PROGRAM MAIN
VAR
	SealedinCoil: FbSealedinCoil;
	xTrigger: BOOL;
	xSealedInCoil: BOOL;
	StateCoilFaultCoil: FbStateCoilFaultCoil;
	xBreakCondition: BOOL;
	xMemoryCoil: BOOL;
	StartStopCircuit: FbStartStopCircuit;
	xStart: BOOL;
	xStop: BOOL;
	/// use SR instead 
	SetReset: FbSetReset;
	xRun: BOOL;
	xSet: BOOL;
	/// use RS instead 
	ResetSet: FbResetSet;
	xReset: BOOL;
	xQs: BOOL;
	xQr: BOOL;
	/// use BLINK instead 
	Flasher: FbFlasher;
	xFlashingLight: BOOL;
	Debounce: FbDebounce;
	xInput: BOOL;
	xInputDebounced: BOOL;
	ExtendCylinder: fbStep;
	xExtendCylinderCmd: BOOL;
	TONExtendCylinderDone: TON;
	xExtendCylinderDone: BOOL;
	tETExtend: TIME;
	RetractCylinder: fbStep;
	xRetractCylinderCmd: BOOL;
	TONRetractCylinderDone: TON;
	tETRetract: TIME;
	Mission: FbMission;
	xMission1Start: BOOL;
	xMission2Start: BOOL;
	xMission1Done: BOOL;
	xMission2Done: BOOL;
	xNoMission: BOOL;
	xMission1Busy: BOOL;
	xMission2Busy: BOOL;
	FiveRung: fbFiveRung;
	xFromSeqLogic: BOOL;
	xEStopOK: BOOL;
	xAutoMode: BOOL;
	xManMode: BOOL;
	xPushButton: BOOL;
	xSensor: BOOL;
	xResetFault: BOOL;
	xTriggerf: BOOL;
	xSafe: BOOL;
	xCommand: BOOL;
	xInPosition: BOOL;
	xTimeoutFault: BOOL;
	Mode: FbMode;
	xAutoModePB: BOOL;
	xManModePB: BOOL;
	xAutoSelected: BOOL;
	xManualSelected: BOOL;
END_VAR

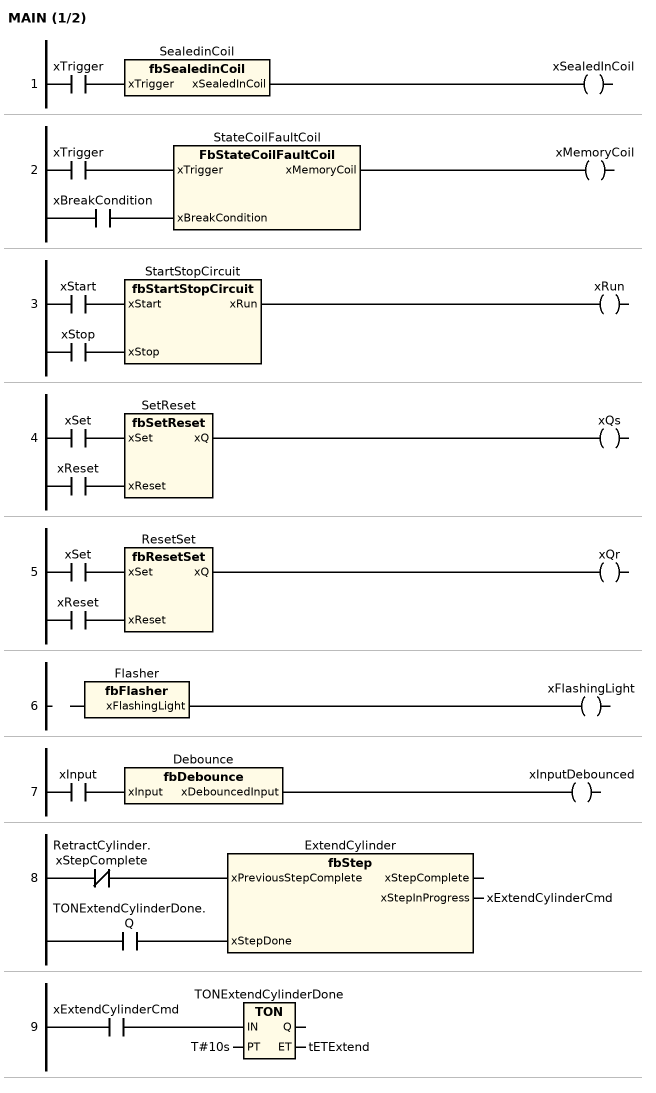
// NETWORK 1
SealedinCoil(xTrigger := xTrigger); // fbSealedinCoil
xSealedInCoil := SealedinCoil.xSealedInCoil;

// NETWORK 2
StateCoilFaultCoil(xTrigger := xTrigger, xBreakCondition := xBreakCondition); // FbStateCoilFaultCoil
xMemoryCoil := StateCoilFaultCoil.xMemoryCoil;

// NETWORK 3
StartStopCircuit(xStart := xStart, xStop := xStop); // fbStartStopCircuit
xRun := StartStopCircuit.xRun;

// NETWORK 4
SetReset(xSet := xSet, xReset := xReset); // fbSetReset
xQs := SetReset.xQ;

// NETWORK 5
ResetSet(xSet := xSet, xReset := xReset); // fbResetSet
xQr := ResetSet.xQ;

// NETWORK 6
Flasher(); // fbFlasher
xFlashingLight := Flasher.xFlashingLight;

// NETWORK 7
Debounce(xInput := xInput); // fbDebounce
xInputDebounced := Debounce.xDebouncedInput;

// NETWORK 8
ExtendCylinder(
    xPreviousStepComplete := NOT RetractCylinder.xStepComplete,
    xStepDone := TONExtendCylinderDone.Q,
    xStepInProgress => xExtendCylinderCmd); // fbStep

// NETWORK 9
TONExtendCylinderDone(IN := xExtendCylinderCmd, PT := T#10s, ET => tETExtend); // TON

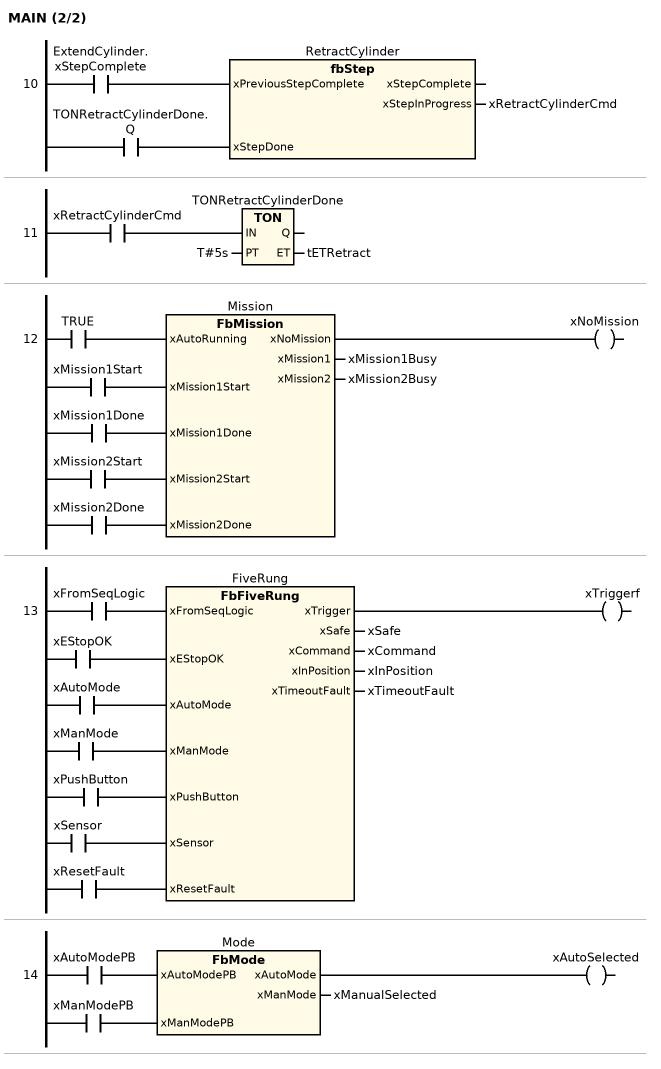
// NETWORK 10
RetractCylinder(
    xPreviousStepComplete := ExtendCylinder.xStepComplete,
    xStepDone := TONRetractCylinderDone.Q,
    xStepInProgress => xRetractCylinderCmd); // fbStep

// NETWORK 11
TONRetractCylinderDone(IN := xRetractCylinderCmd, PT := T#5s, ET => tETRetract); // TON

// NETWORK 12
Mission(
    xAutoRunning := TRUE,
    xMission1Start := xMission1Start,
    xMission1Done := xMission1Done,
    xMission2Start := xMission2Start,
    xMission2Done := xMission2Done,
    xMission1 => xMission1Busy,
    xMission2 => xMission2Busy); // FbMission
xNoMission := Mission.xNoMission;

// NETWORK 13
FiveRung(
    xFromSeqLogic := xFromSeqLogic,
    xEStopOK := xEStopOK,
    xAutoMode := xAutoMode,
    xManMode := xManMode,
    xPushButton := xPushButton,
    xSensor := xSensor,
    xResetFault := xResetFault,
    xSafe => xSafe,
    xCommand => xCommand,
    xInPosition => xInPosition,
    xTimeoutFault => xTimeoutFault); // FbFiveRung
xTriggerf := FiveRung.xTrigger;

// NETWORK 14
Mode(xAutoModePB := xAutoModePB, xManModePB := xManModePB, xManMode => xManualSelected); // FbMode
xAutoSelected := Mode.xAutoMode;

END_PROGRAM

(* stored: Version 1.1.0.1, ProductVersion 3.1.4024.12
   POU MAIN: Id {fceb3a4a-488b-45f3-81c1-d253e50a3c0f}, SpecialFunc None *)
